KUKA KRL data list: DEMO_MAIN3.dat

&ACCESS RVP
&REL 9
&COMMENT Main03
&PARAM DISKPATH = KRC:\R1\Program\PlcDemo
DEFDAT  DEMO_MAIN3
;FOLD EXTERNAL DECLARATIONS;%{PE}%MKUKATPBASIS,%CEXT,%VCOMMON,%P
;FOLD BASISTECH EXT;%{PE}%MKUKATPBASIS,%CEXT,%VEXT,%P
EXT  BAS (BAS_COMMAND  :IN,REAL  :IN )
DECL INT SUCCESS
;ENDFOLD (BASISTECH EXT)
;FOLD USER EXT;%{E}%MKUKATPUSER,%CEXT,%VEXT,%P
;Make your modifications here

;ENDFOLD (USER EXT)
;ENDFOLD (EXTERNAL DECLARATIONS)
DECL MODULEPARAM_T LAST_TP_PARAMS={PARAMS[] "PLC.PROGNO=3  "}
ENDDAT
